PROGRAM INIT
VAR
	MC_MoveAbsolute_1 : MC_MoveAbsolute;
	MC_MoveAbsolute_2 : MC_MoveAbsolute;
	MC_MoveAbsolute_3 : MC_MoveAbsolute;
	MC_MoveAbsolute_4 : MC_MoveAbsolute;
	MC_MoveAbsolute_5 : MC_MoveAbsolute;
	MC_MoveAbsolute_6 : MC_MoveAbsolute;
END_VAR

MC_MoveAbsolute_1(
	Axis:= AXIS.Axis1, 
	Execute:= INIT_Execute1, 
	Position:= , 
	Velocity:= , 
	Acceleration:= , 
	Deceleration:= , 
	Jerk:= , 
	BufferMode:= , 
	Options:= , 
	Done=> , 
	Busy=> , 
	Active=> , 
	CommandAborted=> , 
	Error=> , 
	ErrorID=> );
	
MC_MoveAbsolute_2(
	Axis:= AXIS.Axis2, 
	Execute:= INIT_Execute2, 
	Position:= , 
	Velocity:= , 
	Acceleration:= , 
	Deceleration:= , 
	Jerk:= , 
	BufferMode:= , 
	Options:= , 
	Done=> , 
	Busy=> , 
	Active=> , 
	CommandAborted=> , 
	Error=> , 
	ErrorID=> );
	
MC_MoveAbsolute_3(
	Axis:= AXIS.Axis3, 
	Execute:= INIT_Execute3, 
	Position:= , 
	Velocity:= , 
	Acceleration:= , 
	Deceleration:= , 
	Jerk:= , 
	BufferMode:= , 
	Options:= , 
	Done=> , 
	Busy=> , 
	Active=> , 
	CommandAborted=> , 
	Error=> , 
	ErrorID=> );
	
MC_MoveAbsolute_4(
	Axis:= AXIS.Axis4, 
	Execute:= INIT_Execute4, 
	Position:= , 
	Velocity:= , 
	Acceleration:= , 
	Deceleration:= , 
	Jerk:= , 
	BufferMode:= , 
	Options:= , 
	Done=> , 
	Busy=> , 
	Active=> , 
	CommandAborted=> , 
	Error=> , 
	ErrorID=> );
	
MC_MoveAbsolute_5(
	Axis:= AXIS.Axis5, 
	Execute:= INIT_Execute5, 
	Position:= , 
	Velocity:= , 
	Acceleration:= , 
	Deceleration:= , 
	Jerk:= , 
	BufferMode:= , 
	Options:= , 
	Done=> , 
	Busy=> , 
	Active=> , 
	CommandAborted=> , 
	Error=> , 
	ErrorID=> );
	
MC_MoveAbsolute_6(
	Axis:= AXIS.Axis6, 
	Execute:= INIT_Execute6, 
	Position:= , 
	Velocity:= , 
	Acceleration:= , 
	Deceleration:= , 
	Jerk:= , 
	BufferMode:= , 
	Options:= , 
	Done=> , 
	Busy=> , 
	Active=> , 
	CommandAborted=> , 
	Error=> , 
	ErrorID=> );

END_PROGRAM

(* stored: Version 1.1.0.1, ProductVersion 3.1.4024.0
   POU INIT: Id {5b8a4dc9-f9fa-493c-8b10-dafd47b6e3d9}, SpecialFunc None *)
